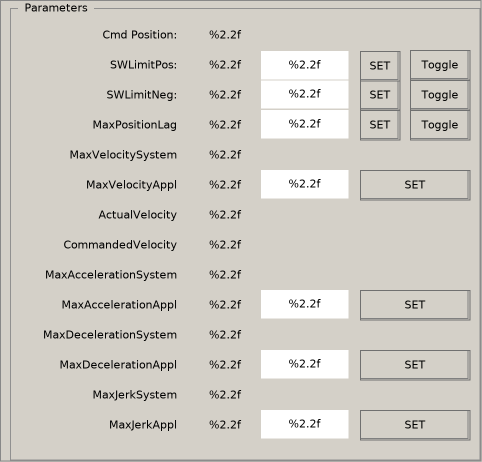
VISUALIZATION Parameters  // 482x462
    GroupBox (10,0 470x460), "Parameters"
        Textfield (170,20 90x30), "%2.2f", text variable: GVL.axes[MAIN.hmiAxisSelect].fParameters[1]
        Textfield (10,50 160x30), "SWLimitPos:"
        Textfield (10,20 160x30), "Cmd Position:"
        Textfield (170,50 90x30), "%2.2f", text variable: GVL.axes[MAIN.hmiAxisSelect].fParameters[2], input disabled if: NOT GVL.axes[MAIN.hmiAxisSelect].bSoftLimPosEn
        Textfield (170,80 90x30), "%2.2f", text variable: GVL.axes[MAIN.hmiAxisSelect].fParameters[3], input disabled if: NOT GVL.axes[MAIN.hmiAxisSelect].bSoftLimNegEn
        Textfield (250,79 89x30), "%2.2f", text variable: GVL.SwLimitNeg
            OnMouseClick: write GVL.SwLimitNeg via Default
        Button (350,80 40x30), "SET"
            toggle GVL.axes[MAIN.hmiAxisSelect].bEXECUTE
            OnMouseClick: execute {
                GVL.axes[Main.hmiAxisSelect].eCommand:=eMcCommand.WriteParameter;
                GVL.axes[Main.hmiAxisSelect].fParameterValue:=GVL.SwLimitNeg;
                GVL.axes[Main.hmiAxisSelect].iParameterIndex:=eRWParameter.SWLimitNeg;
                GVL.axes[Main.hmiAxisSelect].bExecute:=TRUE;
            }
        Button (400,50 60x30), "Toggle", pressed state: GVL.axes[MAIN.hmiAxisSelect].bSoftLimPosEn, text list: 'ButtonStates', text index: GVL.axes[MAIN.hmiAxisSelect].bSoftLimPosEn
            toggle GVL.axes[MAIN.hmiAxisSelect].bEXECUTE
            OnMouseClick: execute {
                GVL.axes[MAIN.hmiAxisSelect].bInput:=NOT GVL.axes[MAIN.hmiAxisSelect].bSoftLimPosEn;
                GVL.axes[MAIN.hmiAxisSelect].eCommand:=eMcCommand.WriteBoolParameter;
                GVL.axes[MAIN.hmiAxisSelect].iParameterIndex:=eRWParameter.EnableLimitPos;
                GVL.axes[MAIN.hmiAxisSelect].bExecute:=TRUE;
            }
        Button (400,80 60x30), "Toggle", pressed state: GVL.axes[MAIN.hmiAxisSelect].bSoftLimNegEn, text list: 'ButtonStates', text index: GVL.axes[MAIN.hmiAxisSelect].bSoftLimNegEn
            toggle GVL.axes[MAIN.hmiAxisSelect].bEXECUTE
            OnMouseClick: execute {
                GVL.axes[MAIN.hmiAxisSelect].bInput:=NOT GVL.axes[MAIN.hmiAxisSelect].bSoftLimNegEn;
                GVL.axes[MAIN.hmiAxisSelect].eCommand:=eMcCommand.WriteBoolParameter;
                GVL.axes[MAIN.hmiAxisSelect].iParameterIndex:=eRWParameter.EnableLimitNeg;
                GVL.axes[MAIN.hmiAxisSelect].bExecute:=TRUE;
            }
        Textfield (10,110 160x30), "MaxPositionLag"
        Textfield (10,140 160x30), "MaxVelocitySystem"
        Textfield (10,170 160x30), "MaxVelocityAppl"
        Textfield (10,200 160x30), "ActualVelocity"
        Textfield (10,230 160x30), "CommandedVelocity"
        Textfield (170,260 90x30), "%2.2f", text variable: GVL.axes[MAIN.hmiAxisSelect].fParameters[12]
        Textfield (10,290 160x30), "MaxAccelerationAppl"
        Textfield (10,320 160x30), "MaxDecelerationSystem"
        Textfield (10,380 160x30), "MaxJerkSystem"
        Button (350,51 40x30), "SET"
            toggle GVL.axes[MAIN.hmiAxisSelect].bEXECUTE
            OnMouseClick: execute {
                GVL.axes[Main.hmiAxisSelect].eCommand:=eMcCommand.WriteParameter;
                GVL.axes[Main.hmiAxisSelect].fParameterValue:=GVL.SwLimitPos;
                GVL.axes[Main.hmiAxisSelect].iParameterIndex:=eRWParameter.SWLimitPos;
                GVL.axes[Main.hmiAxisSelect].bExecute:=TRUE;
            }
        Textfield (10,80 160x30), "SWLimitNeg:"
        Textfield (170,110 90x30), "%2.2f", text variable: GVL.axes[MAIN.hmiAxisSelect].fParameters[7], input disabled if: NOT GVL.axes[MAIN.hmiAxisSelect].bPosLagEn
        Textfield (250,109 89x30), "%2.2f", text variable: GVL.MaxPositionLag
            OnMouseClick: write GVL.MaxPositionLag via Default
        Button (350,110 40x30), "SET"
            toggle GVL.axes[MAIN.hmiAxisSelect].bEXECUTE
            OnMouseClick: execute {
                GVL.axes[Main.hmiAxisSelect].eCommand:=eMcCommand.WriteParameter;
                GVL.axes[Main.hmiAxisSelect].fParameterValue:=GVL.MaxPositionLag;
                GVL.axes[Main.hmiAxisSelect].iParameterIndex:=eRWParameter.MaxPositionLag;
                GVL.axes[Main.hmiAxisSelect].bExecute:=TRUE;
            }
        Button (400,110 60x30), "Toggle", pressed state: GVL.axes[MAIN.hmiAxisSelect].bPosLagEn, text list: 'ButtonStates', text index: GVL.axes[MAIN.hmiAxisSelect].bPosLagEn
            toggle GVL.axes[MAIN.hmiAxisSelect].bEXECUTE
            OnMouseClick: execute {
                GVL.axes[MAIN.hmiAxisSelect].bInput:=NOT GVL.axes[MAIN.hmiAxisSelect].bPosLagEn;
                GVL.axes[MAIN.hmiAxisSelect].eCommand:=eMcCommand.WriteBoolParameter;
                GVL.axes[MAIN.hmiAxisSelect].iParameterIndex:=eRWParameter.EnablePosLagMonitoring;
                GVL.axes[MAIN.hmiAxisSelect].bExecute:=TRUE;
            }
        Textfield (170,140 90x30), "%2.2f", text variable: GVL.axes[MAIN.hmiAxisSelect].fParameters[8]
        Textfield (170,170 90x30), "%2.2f", text variable: GVL.axes[MAIN.hmiAxisSelect].fParameters[9]
        Textfield (250,169 89x30), "%2.2f", text variable: GVL.MaxVelocityAppl
            OnMouseClick: write GVL.MaxVelocityAppl via Default
        Button (350,170 110x30), "SET"
            toggle GVL.axes[MAIN.hmiAxisSelect].bEXECUTE
            OnMouseClick: execute {
                GVL.axes[Main.hmiAxisSelect].eCommand:=eMcCommand.WriteParameter;
                GVL.axes[Main.hmiAxisSelect].fParameterValue:=GVL.MaxVelocityAppl;
                GVL.axes[Main.hmiAxisSelect].iParameterIndex:=eRWParameter.MaxVelocityAppl;
                GVL.axes[Main.hmiAxisSelect].bExecute:=TRUE;
            }
        Textfield (170,200 90x30), "%2.2f", text variable: GVL.axes[MAIN.hmiAxisSelect].fParameters[10]
        Textfield (170,230 90x30), "%2.2f", text variable: GVL.axes[MAIN.hmiAxisSelect].fParameters[11]
        Textfield (10,260 160x30), "MaxAccelerationSystem"
        Textfield (170,290 90x30), "%2.2f", text variable: GVL.axes[MAIN.hmiAxisSelect].fParameters[13]
        Textfield (250,289 89x30), "%2.2f", text variable: GVL.MaxAccelerationAppl
            OnMouseClick: write GVL.MaxAccelerationAppl via Default
        Button (350,290 110x30), "SET"
            toggle GVL.axes[MAIN.hmiAxisSelect].bEXECUTE
            OnMouseClick: execute {
                GVL.axes[Main.hmiAxisSelect].eCommand:=eMcCommand.WriteParameter;
                GVL.axes[Main.hmiAxisSelect].fParameterValue:=GVL.MaxAccelerationAppl;
                GVL.axes[Main.hmiAxisSelect].iParameterIndex:=eRWParameter.MaxAccelerationAppl;
                GVL.axes[Main.hmiAxisSelect].bExecute:=TRUE;
            }
        Textfield (170,320 90x30), "%2.2f", text variable: GVL.axes[MAIN.hmiAxisSelect].fParameters[14]
        Textfield (10,350 160x30), "MaxDecelerationAppl"
        Textfield (170,350 90x30), "%2.2f", text variable: GVL.axes[MAIN.hmiAxisSelect].fParameters[15]
        Textfield (250,349 89x30), "%2.2f", text variable: GVL.MaxDecelerationAppl
            OnMouseClick: write GVL.MaxDecelerationAppl via Default
        Button (350,350 110x30), "SET"
            toggle GVL.axes[MAIN.hmiAxisSelect].bEXECUTE
            OnMouseClick: execute {
                GVL.axes[Main.hmiAxisSelect].eCommand:=eMcCommand.WriteParameter;
                GVL.axes[Main.hmiAxisSelect].fParameterValue:=GVL.MaxDecelerationAppl;
                GVL.axes[Main.hmiAxisSelect].iParameterIndex:=eRWParameter.MaxDecelerationAppl;
                GVL.axes[Main.hmiAxisSelect].bExecute:=TRUE;
            }
        Textfield (170,380 90x30), "%2.2f", text variable: GVL.axes[MAIN.hmiAxisSelect].fParameters[16]
        Textfield (10,410 160x30), "MaxJerkAppl"
        Textfield (170,410 90x30), "%2.2f", text variable: GVL.axes[MAIN.hmiAxisSelect].fParameters[17]
        Textfield (250,409 89x30), "%2.2f", text variable: GVL.MaxJerkAppl
            OnMouseClick: write GVL.MaxJerkAppl via Default
        Button (350,410 110x30), "SET"
            toggle GVL.axes[MAIN.hmiAxisSelect].bEXECUTE
            OnMouseClick: execute {
                GVL.axes[Main.hmiAxisSelect].eCommand:=eMcCommand.WriteParameter;
                GVL.axes[Main.hmiAxisSelect].fParameterValue:=GVL.MaxJerkAppl;
                GVL.axes[Main.hmiAxisSelect].iParameterIndex:=eRWParameter.MaxJerkAppl;
                GVL.axes[Main.hmiAxisSelect].bExecute:=TRUE;
            }
        Textfield (250,50 89x30), "%2.2f", text variable: GVL.SwLimitPos
            OnMouseClick: write GVL.SwLimitPos via Default
END_VISUALIZATION

(* stored: Version 1.1.0.1, ProductVersion 3.1.4022.12
   Visu Parameters: Id {6f2fabd5-25a4-4dfe-b86f-3cd159b0d0fe} *)
